{attribute 'qualified_only'}
{attribute 'strict'}
{attribute 'to_string'}
TYPE E_Request :
(
	{attribute 'hide'}
    Undefined   := 0,
	Reset       := 1,
    Start       := 2,
    Pause       := 4,	
    Hold      	:= 8,
	Complete	:= 16,	
    Stop        := 32,
	Abort       := 64
);
END_TYPE

(* stored: Version 1.1.0.1
   DUT E_Request: Id {d3b20770-b5da-468b-8276-148bae048ad0} *)
